// TIA Portal V21 export
DATA_BLOCK "PRINTING_1"   // DB193
{ S7_Optimized_Access := 'FALSE' }
// stored: AutoNumber false
   VAR
      L1 : String[80] := '                  M/s. LABORATE PHARMACEUTICALS INDIA LIMITED             ';
      L2 : String[80] := '               111, YAMUNA NAGAR ROAD, SATIWALA, PAONTA SAHIB,         ';
      L3 : String[80] := '               DISS.- SIRMOUR, HIMACHAL PRADESH - 173025 INDIA';
      L4 : String[80] := '              STERILIZING DEPYROGENATION TUNNEL (MODEL NO- SDT-C-5H)    ';
      L5 : String[80] := '              ----------------------------------------------------------';
      L6 : String[80] := '  EQUIPMENT ID        :';
      L7 : String[80] := '  PRODUCT NAME        :';
      L8 : String[80] := '  BATCH NO            :';
      L9 : String[80] := '                                                             DATE:  /  /       ';
      L10 : String[80] := '  PROCESS STARTED AT  :   :  :     ';
      L11 : String[80] := '  OPERATOR NAME       :';
      L12 : String[80] := '  TUNNEL MODE         :';
      L13 : String[80] := '  RECEIPE TYPE        :';
      L14 : String[80] := '-------------------------------------------------------------------------';
      L15 : String[80] := '  CONTROL TEMP (DEG.C)    :                   CONVEYOR SPEED (mm/min)   :     ';
      L16 : String[80] := '  CONVEYOR ON TEMP (DEG.C):                   CONVEYOR OFF TEMP (DEG.C) :    ';
      L17 : String[80] := '  SHUTDOWN TEMP (DEG.C)   :                   PRINTING INTERVAL (SEC)   :       ';
      L18 : String[80] := '                                            ';
      L19 : String[80] := '  CHECKED BY:                                 VERIFIED BY:';
      L20 : String[80] := '********************************************************************************';
      L21 : String[80] := '  DZ=DRYING ZONE            MHZ=MAIN HEATING ZONE   ST IN=STERILIZATION IN';
      L22 : String[80] := '  ST OUT=STERILIZATION OUT  CZ UP=COOLING ZONE UP   CZ DOWN=COOLING ZONE DOWN ';
      L23 : String[80] := '********************************************************************************';
      L24 : String[80] := '             :  CH-1  :  CH-2  :  CH-3  :  CH-4  :  CH-5  :  CH-6  :  CONVEYOR  ';
      L25 : String[90] := '     TIME    :  DZ    :  MHZ   :  ST IN :  ST OUT:  CZ UP :  CZDOWN:  SPEED ';
      L26 : String[80] := '             :  DEG.C :  DEG.C :  DEG.C :  DEG.C :  DEG.C :  DEG.C :  mm/min ';
      L27 : String[80] := '--------------------------------------------------------------------------------';
      L28 : String[80] := '    :  :                                                                     ';
      L29 : String[80] := '                                                                     ';
      L30 : String[80];
      L31 : String[80] := '               RECEIPE TYPE :                                                   ';
      L32 : String[80] := '--------------------------------------------------------------------------------';
      ALM1 : String[80] := '    :  :       EMERGENCY PRESSED ';
      ALM2 : String[80] := '    :  :       TURBIN VFD TRIP ';
      ALM3 : String[80] := '    :  :       CONVEYOR SUPPLY FAIL ';
      ALM4 : String[80] := '    :  :       LAF SUPPLY FAIL ';
      ALM5 : String[80] := '    :  :       TURBIN SUPPLY FAIL';
      ALM6 : String[80] := '    :  :       VAPOR EXHAUST SUPPLY FAIL';
      ALM7 : String[80] := '    :  :       HEATER SUPPLY FAIL';
      ALM8 : String[80] := '    :  :       TEMPERATURE OVERSHOOT';
      ALM9 : String[80] := '    :  :       VAPOUR EXHAUST TRIP';
      ALM10 : String[80] := '    :  :       SINGLE PHASE FAIL ';
      ALM11 : String[80] := '    :  :       DRYING ZONE PRESSURE LOW/PLEASE CHECK SENSOR OR BLOWER ';
      ALM12 : String[80] := '    :  :       COOLING ZONE PRESSURE LOW/PLEASE CHECK SENSOR OR BLOWER ';
      ALM13 : String[80] := '    :  :       STERILIZING  PREESURE LOW/PLEASE CHECK SENSOR OR TURBINE ';
      ALM14 : String[80] := '    :  :       CONVEYOR VFD OVERLOAD ';
      ALM15 : String[80] := '    :  :       MAIN HEAT RTD SENSOR FAIL ';
      ALM16 : String[80] := '    :  :       STERILE IN RTD SENSOR FAIL ';
      ALM17 : String[80] := '    :  :       STERILE OUT RTD SENSOR FAIL ';
      ALM18 : String[80] := '    :  :       CONVEYOR VFD TRIP ';
      ALM19 : String[80] := '    :  :       SHUTDOWN CYCLE STARTED ';
      ALM20 : String[80] := '    :  :                     *****PROCESS COMPLETED*****';
      ALM21 : String[80] := '  CHECKED BY:                                 VERIFIED BY:';
      "BATCH SIZE" : String[80] := '  BATCH SIZE          :';
      "CONTAINER SIZE" : String[80] := '  CONTAINER SIZE      :';
      "BLANK LINE" : String[80] := '                                                                ';
      ADDRESS : String[80] := ' ';
   END_VAR
BEGIN
END_DATA_BLOCK
